// TIA Portal V20 export
DATA_BLOCK "BK16"   // DB260
// stored: MemoryReserve 100
   VAR
      "X10-1 FINAL VISION STAGE LIFT UP" : Bool;
      "X10-2 FINAL VISION STAGE LIFT DOWN" : Bool;
      "X12-1 FINAL VISION LIGHT UP" : Bool;
      "X12-2 FINAL VISION LIGHT DOWN" : Bool;
      "X14-1 FINAL VISION STAGE DETECT SENSOR" : Bool;
      "X14-2 SPARE" : Bool;
      "X16-1 SPARE" : Bool;
      "X16-2 SPARE" : Bool;
   END_VAR
BEGIN
END_DATA_BLOCK
